FUNCTION_BLOCK SYSFS_IO (* Service Interface Function Block Type *)
  (* Standard: 61499-2 *)
  (* Version 0.0, 17/02/2021, SESA515713, nxtControl GmBH, template *)
  PACKAGE Flexbridge.Iceblock;
  (* Compiler Cpp nxtControl builtin 1.0 *)
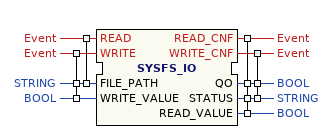
  EVENT_INPUT
    READ WITH FILE_PATH; (* Service Initialization *)
    WRITE WITH FILE_PATH, WRITE_VALUE; (* Service Request *)
  END_EVENT
  EVENT_OUTPUT
    READ_CNF WITH QO, STATUS, READ_VALUE; (* Initialization Confirm *)
    WRITE_CNF WITH QO, STATUS; (* Confirmation of Requested Service *)
  END_EVENT
  VAR_INPUT
    FILE_PATH : STRING; (* Event Input Qualifier *)
    WRITE_VALUE : BOOL; (* Service Parameters *)
  END_VAR
  VAR_OUTPUT
    QO : BOOL;
    STATUS : STRING;
    READ_VALUE : BOOL; (* Service Status *)
  END_VAR
  SERVICE SYSFS_IO/RESOURCE
    SEQUENCE normal_establishment
      SYSFS_IO.READ+(WRITE_VALUE) -> RESOURCE.initialize(WRITE_VALUE) -> SYSFS_IO.READ_CNF+();
    END_SEQUENCE
    SEQUENCE unsuccessful_establishment
      SYSFS_IO.READ+(WRITE_VALUE) -> RESOURCE.initialize(WRITE_VALUE) -> SYSFS_IO.READ_CNF-(READ_VALUE);
    END_SEQUENCE
    SEQUENCE request_confirm
      SYSFS_IO.WRITE+(SD) -> RESOURCE.request(SD) -> SYSFS_IO.WRITE_CNF+(RD);
    END_SEQUENCE
    SEQUENCE request_inhibited
      SYSFS_IO.WRITE-(SD) -> SYSFS_IO.WRITE_CNF-(READ_VALUE);
    END_SEQUENCE
    SEQUENCE request_error
      SYSFS_IO.WRITE+(SD) -> RESOURCE.request(SD) -> SYSFS_IO.WRITE_CNF-(READ_VALUE);
    END_SEQUENCE
    SEQUENCE indication_response
      RESOURCE.indicate(RD) -> SYSFS_IO.IND+(RD);
      SYSFS_IO.RSP(FILE_PATH,SD) -> RESOURCE.response(FILE_PATH,SD);
    END_SEQUENCE
    SEQUENCE indication_inhibited
      RESOURCE.indicate(RD,FILE_PATH=FALSE) -> RESOURCE.inhibited();
    END_SEQUENCE
    SEQUENCE error_indication
      RESOURCE.error(READ_VALUE) -> SYSFS_IO.IND-(READ_VALUE);
    END_SEQUENCE
    SEQUENCE application_initiated_termination
      SYSFS_IO.READ-() -> RESOURCE.terminate() -> SYSFS_IO.READ_CNF-(READ_VALUE);
    END_SEQUENCE
    SEQUENCE resource_initiated_termination
      -> SYSFS_IO.READ_CNF-(READ_VALUE);
    END_SEQUENCE
  END_SERVICE
END_FUNCTION_BLOCK
